// SIMATIC S7-200 project (STEP 7-Micro/WIN), CPU 221 REL 01.10

SYMBOL_TABLE USER1
start            I0.0
estop            I0.1
BT1              Q0.0
BT2              Q0.1
END_SYMBOL_TABLE

ORGANIZATION_BLOCK MAIN:OB1
TITLE=PROGRAM COMMENTS
BEGIN
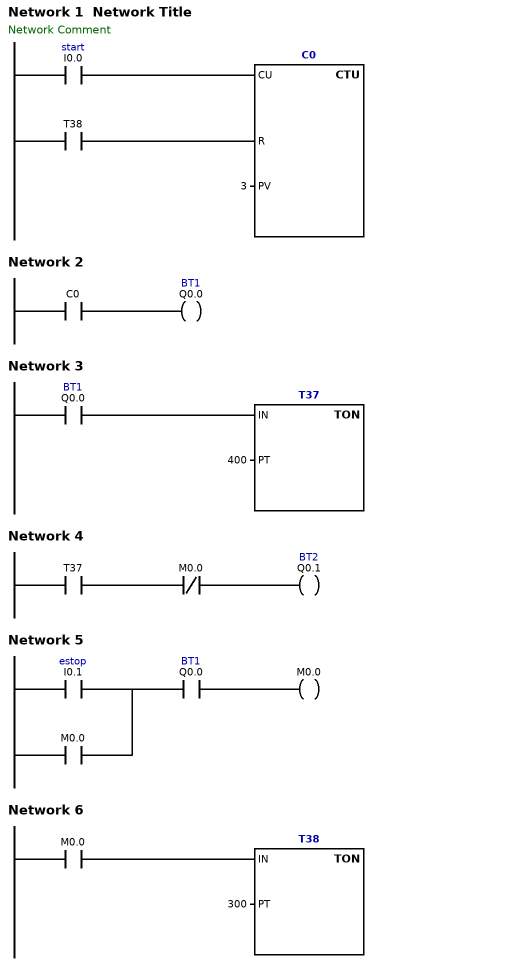
Network 1 // Network Title
// Network Comment
LD     start:I0.0
LD     T38
CTU    C0, 3
Network 2
LD     C0
=      BT1:Q0.0
Network 3
LD     BT1:Q0.0
TON    T37, 400
Network 4
LD     T37
AN     M0.0
=      BT2:Q0.1
Network 5
LD     estop:I0.1
O      M0.0
A      BT1:Q0.0
=      M0.0
Network 6
LD     M0.0
TON    T38, 300
END_ORGANIZATION_BLOCK
